# EPICS substitutions: NFIPM/NFIPM-IOC-01App/db/motor.substitutions
file $(MOTOR)/db/motor.db {
pattern {P,    M,         DTYP,      DESC,   EGU,  DIR,  VELO,  VBAS, ACCL, BDST, BVEL, BACC,    MRES,    ERES, UEIP, PREC, DHLM, DLLM, INIT, C, S, OFF }
{"\$(P)", "\$(M)", "PMNC87xx", "\$(NAME) (New Focus)",    "\$(EGU)",  "Pos",  "\$(VELO)",   "\$(VBAS)",  "\$(ACCL)",    0,    1,   0,   "\$(MRES)",   "\$(ERES)", "\$(UEIP)",    3,   "\$(DHLM)",   "\$(DLLM)",  "", "\$(C)", "\$(S)"}
}

file $(MOTOR)/db/motor_init_extra.db {
pattern {P, M, OFF, JVEL}
{"\$(P)", "\$(M)", "\$(OFF)", "\$(JVEL)"}
}

file $(MOTOR)/db/periodic_polling.db {
pattern {P, M}
{"\$(P)", "\$(M)"}
}
